TYPE ST_BI1Statuses :
STRUCT
END_STRUCT
END_TYPE

(* stored: Version 1.1.0.1, ProductVersion 3.1.4024.0
   DUT ST_BI1Statuses: Id {f2430048-ed8e-037a-272e-19f1b239ad1a} *)
